// TwinCAT 3 PLC project Untitled1
// ProgramVersion: 3.1.4023.0
// libraries:
//   Tc2_Standard, * (Beckhoff Automation GmbH)
//   Tc2_System, * (Beckhoff Automation GmbH)
//   Tc3_Module, * (Beckhoff Automation GmbH)
// project tree:
//   / PlcTask.TcTTO
//   POUs/ MAIN.TcPOU
// real-time tasks:
//   TASK PlcTask: cycle T#10ms, priority 20, ADS port 350

CONFIGURATION Untitled1
    RESOURCE PLC ON TwinCAT3
        TASK PlcTask(INTERVAL := T#10ms, PRIORITY := 20);
        PROGRAM MAIN WITH PlcTask : MAIN;
    END_RESOURCE
END_CONFIGURATION

// ---- POUs/MAIN.TcPOU
PROGRAM MAIN
VAR
	I_StartButton: BOOL;
	I_StopButton: BOOL;
	Q_MotorRun: BOOL;
	tonContactor: TON;
	Q_Star: BOOL;
	Q_Delta: BOOL;
END_VAR

IF I_StartButton THEN
	Q_MotorRun := TRUE;
ELSIF I_StopButton THEN
	Q_MotorRun := FALSE;
END_IF

tonContactor(IN:= Q_MotorRun , PT:=T#10S);

Q_Star := Q_MotorRun AND NOT tonContactor.Q;
Q_Delta :=  Q_MotorRun AND NOT tonContactor.Q;

END_PROGRAM
